INTERFACE I_OutputPort EXTENDS I_Disposable, I_EventEmitter, I_Serializable

METHOD PUBLIC Accept
VAR_INPUT
	Visitor : I_OutputPortVisitor;
END_VAR
END_METHOD

PROPERTY PUBLIC Name : T_MAXSTRING
GET
END_GET
END_PROPERTY

END_INTERFACE

(* stored: Version 1.1.0.1, ProductVersion 3.1.4024.12
   Itf I_OutputPort: Id {ee2ad4f0-687d-0acb-0188-96d2063a474f}
   Method Accept: Id {6b9b017c-be5d-076e-1f48-61c0c312dadd}
   Property Name: Id {67c8a939-6cc5-01f4-2443-86e8aa7bc6b0}
   Get Get: Id {87b1c37b-6a0e-0c82-10a0-6e90c455f4d3} *)
